// TIA Portal V17 export
// export: Created 2024-08-07T21:44:04.6396761Z, ExportSetting WithDefaults, DisplayName Totally Integrated Automation Portal, DisplayVersion V17 Update 7, DisplayName TIA Portal Openness, DisplayVersion V17 Update 7, DisplayName TIA Portal Version Control Interface, DisplayVersion V17, DisplayName SINAMICS Startdrive Advanced, DisplayVersion V17 SP2, DisplayName SINAMICS Startdrive G110M, G120, G120C, G120D, G120P, G115D, DisplayVersion V17 SP2, DisplayName SINAMICS Startdrive G130, G150, S120, S150, SINAMICS MV, S210, DisplayVersion V17 SP2, DisplayName STEP 7 Professional, DisplayVersion V17 Update 7, DisplayName STEP 7 Safety, DisplayVersion V17 Update 6, DisplayName WinCC Advanced / Unified PC, DisplayVersion V17 Update 7
DATA_BLOCK "St1Insertion"   // DB15
{ S7_Optimized_Access := 'TRUE' }
VERSION : 0.1
// stored: AutoNumber true, DBAccessibleFromOPCUA true, DBAccessibleFromWebserver true, IsOnlyStoredInLoadMemory false, IsRetainMemResEnabled false, IsWriteProtectedInAS false, MemoryReserve 100
   VAR
      ExpectedSensors : Array[0..20] of Bool;
      UsedSensors : Array[0..20] of Bool;
      SensorsState : Array[0..20] of Bool;
      SensorsNOK : Array[0..20] of Bool;
      NOKList : Array[0..20] of Int;
      InsertionOK : Bool := TRUE;
      InsertionNOK : Bool := FALSE;
      InsertionEmpty : Bool := TRUE;
      EmptyBits : Array[0..20] of Bool;
      FullBits : Array[0..20] of Bool;
   END_VAR
BEGIN
   ExpectedSensors[0..20] := FALSE;
   UsedSensors[0..20] := FALSE;
   SensorsState[0..20] := FALSE;
   SensorsNOK[0..20] := FALSE;
   NOKList[0..20] := 0;
   EmptyBits[0..20] := FALSE;
   FullBits[0] := FALSE;
   FullBits[1..17] := TRUE;
   FullBits[18..20] := FALSE;
END_DATA_BLOCK
